{attribute addProperty Name "Pneumatic cyclinder"}
FUNCTION_BLOCK fbPiston EXTENDS TcoCore.TcoComponent IMPLEMENTS IPistonGripper, IPistonHorizontal, IPistonVertical
VAR_INPUT
	iHomePositionSensor : BOOL;
	iWorkPositionSensor : BOOL;	
END_VAR

VAR_OUTPUT
	qHomePositionActuator : BOOL;
	qWorkPositionActuator : BOOL;		
END_VAR

VAR
	{attribute addProperty Activity "moves to home position"}
	_moveHomeTask : fbPistonMoveTask(THIS^, TcoCore.NO.Structure);
	{attribute addProperty Activity "moves to work position"}
	_moveWorkTask : fbPistonMoveTask(THIS^, TcoCore.NO.Structure);
END_VAR

_moveHomeTask(PositionSensor := iHomePositionSensor, MoveToPositionSignal := qHomePositionActuator, InverseSignal := qWorkPositionActuator);
_moveWorkTask(PositionSensor := iWorkPositionSensor, MoveToPositionSignal := qWorkPositionActuator, InverseSignal := qHomePositionActuator);

METHOD Close : TcoCore.ITcoTaskStatus
Close := MoveToHome();
END_METHOD

METHOD PROTECTED Manual
VAR_INPUT
END_VAR
END_METHOD

METHOD MoveDown : TcoCore.ITcoTaskStatus
MoveDown := MoveToHome();
END_METHOD

METHOD MoveLeft : TcoCore.ITcoTaskStatus
MoveLeft := MoveToWork();
END_METHOD

METHOD MoveRight : TcoCore.ITcoTaskStatus
MoveRight := MoveToHome();
END_METHOD

METHOD PROTECTED MoveToHome : TcoCore.ITcoTaskStatus
MoveToHome := THIS^._moveHomeTask.Invoke();
END_METHOD

METHOD PROTECTED MoveToWork : TcoCore.ITcoTaskStatus
MoveToWork := THIS^._moveWorkTask.Invoke();
END_METHOD

METHOD MoveUp : TcoCore.ITcoTaskStatus
MoveUp := MoveToWork();
END_METHOD

METHOD Open : TcoCore.ITcoTaskStatus
Open := MoveToWork();
END_METHOD

METHOD  Restore : ITcoRestorable
THIS^._moveHomeTask.Restore();
THIS^._moveWorkTask.Restore();
END_METHOD

(*~
	<docu>
		<summary>
		    Custom service (manual, maintenance) logic.
			This method must be implemented in derived class.
		</summary>			
	</docu>	
~*)
METHOD PROTECTED  ServiceMode
END_METHOD

END_FUNCTION_BLOCK

(* stored: Version 1.1.0.1, ProductVersion 3.1.4024.9
   POU fbPiston: Id {c4094ed5-4fe0-0f6e-24e6-4cc0fa53181e}, SpecialFunc None
   Folder Gripper: Id {f422736b-a4ff-4bdb-aafe-11613f36e687}
   Folder Horizontal: Id {39838326-8ba7-42ff-93a8-48faae7dd3f1}
   Folder Vertical: Id {223d4b1a-3aa8-49b9-8e25-d72b18672816}
   Method Close: Id {27e35537-09a4-4073-91f1-6d0fb26c5fde}
   Method Manual: Id {e2305248-08d3-0a45-0227-6f8abe0d86d9}
   Method MoveDown: Id {74594fe6-2f16-4e5a-ac52-6a94752e91a6}
   Method MoveLeft: Id {a307d3d0-8d36-45ef-886c-fcf0072551d2}
   Method MoveRight: Id {97b5e4c3-9c2c-4e7c-8dc9-d8033ccc70ac}
   Method MoveToHome: Id {ec08a57d-3edb-01f0-35bc-3c8a96242bb9}
   Method MoveToWork: Id {e9e0be0c-566d-0749-1c75-1097c8dadecf}
   Method MoveUp: Id {f237180e-da3e-47f0-8a14-888f70a71c84}
   Method Open: Id {08e58c4c-094c-457f-abda-3144fa1f4bd8}
   Method Restore: Id {fc7ee28d-fd88-0b69-144e-14e0b2374ab2}
   Method ServiceMode: Id {bfab5335-2802-01ec-2297-5bec2ba8c2d8} *)
